// Mitsubishi GX Works2 project: BookEX3_1 POU   PLC: Q13UDV

TYPE CnvBlock : STRUCT
  bStartSW : BOOL;
  bEndSW : BOOL;
  BoxCnt : ARRAY [0..9] OF INT;
  sName : STRING[32];
  tOnDelay : TIME;
END_STRUCT END_TYPE

TYPE sdtLog : STRUCT
  idMonth : INT;
  idDay : INT;
  idHour : INT;
  idMin : INT;
  idSec : INT;
  idPID : DINT;
  wdData : ARRAY [0..39] OF INT;
  idYear : INT;
  idMsgNo : INT;
  idMsgLeng : INT;
END_STRUCT END_TYPE

TYPE ServoBlk : STRUCT
  RunCode : INT;
  ErrCode : INT;
  WarnCode : INT;
  ServoSts : WORD;
  CmdPos : DINT;
  CurrPos : DINT;
  CurrSp : INT;
  Torque : INT;
END_STRUCT END_TYPE

// global labels: Global
VAR_GLOBAL
  bVar0 AT M5000 : BOOL;
  abArray0 AT M5010 : ARRAY [0..49] OF BOOL;
  sStr0 AT D5000 : STRING[199];
  sStr1 AT D5100 : STRING[199];
  sStr2 AT D5200 : STRING[199];
  sStr3 AT D5300 : STRING[199];
  sStr4 AT D5400 : STRING[199];
  sStr5 AT D5500 : STRING[199];
  sStr6 AT D5600 : STRING[199];
  sStr7 AT D5700 : STRING[199];
  sStr8 AT D5800 : STRING[199];
  sStr9 AT D5900 : STRING[199];
  iVar0 AT D4500 : INT;
  iVar1 AT D4501 : INT;
  iVar2 AT D4502 : INT;
  iVar3 AT D4503 : INT;
  iVar4 AT D4504 : INT;
  iVar5 AT D4505 : INT;
  iVar6 AT D4506 : INT;
  iVar7 AT D4507 : INT;
  iVar8 AT D4508 : INT;
  iVar9 AT D4509 : INT;
  dVar0 AT D4510 : DINT;
  dVar1 AT D4512 : DINT;
  dVar2 AT D4514 : DINT;
  dVar3 AT D4516 : DINT;
  dVar4 AT D4518 : DINT;
  dVar5 AT D4520 : DINT;
  dVar6 AT D4522 : DINT;
  dVar7 AT D4524 : DINT;
  dVar8 AT D4526 : DINT;
  dVar9 AT D4528 : DINT;
  wVar0 AT D4530 : WORD;
  wVar1 AT D4531 : WORD;
  wVar2 AT D4532 : WORD;
  wVar3 AT D4533 : WORD;
  wVar4 AT D4534 : WORD;
  wVar5 AT D4535 : WORD;
  wVar6 AT D4536 : WORD;
  wVar7 AT D4537 : WORD;
  wVar8 AT D4538 : WORD;
  wVar9 AT D4539 : WORD;
  dwVar0 AT D4540 : DWORD;
  dwVar1 AT D4542 : DWORD;
  dwVar2 AT D4544 : DWORD;
  dwVar3 AT D4546 : DWORD;
  dwVar4 AT D4548 : DWORD;
  dwVar5 AT D4550 : DWORD;
  dwVar6 AT D4552 : DWORD;
  dwVar7 AT D4554 : DWORD;
  dwVar8 AT D4556 : DWORD;
  dwVar9 AT D4558 : DWORD;
  fsVar0 AT D4560 : REAL;
  fsVar1 AT D4562 : REAL;
  fsVar2 AT D4564 : REAL;
  fsVar3 AT D4566 : REAL;
  fsVar4 AT D4568 : REAL;
  fsVar5 AT D4570 : REAL;
  fsVar6 AT D4572 : REAL;
  fsVar7 AT D4574 : REAL;
  fsVar8 AT D4576 : REAL;
  fsVar9 AT D4578 : REAL;
  fdVar0 AT D4580 : LREAL;
  tTime0 AT D4620 : TIME;
  tTime1 AT D4622 : TIME;
  tTime2 AT D4624 : TIME;
  tTime3 AT D4626 : TIME;
  tTime4 AT D4628 : TIME;
  tTime5 AT D4630 : TIME;
  tTime6 AT D4632 : TIME;
  tTime7 AT D4634 : TIME;
  tTime8 AT D4636 : TIME;
  tTime9 AT D4638 : TIME;
  tTime10 AT D4640 : TIME;
  bVar1 AT M5001 : BOOL;
  bVar2 AT M5002 : BOOL;
  bVar3 AT M5003 : BOOL;
  bVar4 AT M5004 : BOOL;
  bVar5 AT M5005 : BOOL;
  bVar6 AT M5006 : BOOL;
  bVar7 AT M5007 : BOOL;
  bVar8 AT M5008 : BOOL;
  bVar9 AT M5009 : BOOL;
  abArray1 AT M5060 : ARRAY [0..49] OF BOOL;
  abArray2 AT M5110 : ARRAY [0..49] OF BOOL;
  abArray3 AT M5160 : ARRAY [0..49] OF BOOL;
  abArray4 AT M5210 : ARRAY [0..49] OF BOOL;
  abArray5 AT M5260 : ARRAY [0..49] OF BOOL;
  abArray6 AT M5310 : ARRAY [0..49] OF BOOL;
  abArray7 AT M5360 : ARRAY [0..49] OF BOOL;
  abArray8 AT M5410 : ARRAY [0..49] OF BOOL;
  abArray9 AT M5460 : ARRAY [0..49] OF BOOL;
  fdVar1 AT D4584 : LREAL;
  fdVar2 AT D4588 : LREAL;
  fdVar3 AT D4592 : LREAL;
  fdVar4 AT D4596 : LREAL;
  fdVar5 AT D4600 : LREAL;
  fdVar6 AT D4604 : LREAL;
  fdVar7 AT D4608 : LREAL;
  fdVar8 AT D4612 : LREAL;
  fdVar9 AT D4616 : LREAL;
  aSendData1 AT D100 : ARRAY [0..9] OF INT;
  aiTxData AT D4000 : ARRAY [0..99] OF INT;
  aiRxData AT D4100 : ARRAY [0..99] OF INT;
  iOpenOK AT D3900 : INT;
  iOpenERR AT D3901 : INT;
  iSendOK AT D3902 : INT;
  iSendERR AT D3903 : INT;
  iCloseOK AT D3906 : INT;
  iCloseERR AT D3907 : INT;
  iRecvOK AT D3904 : INT;
  iRecvERR AT D3905 : INT;
  aiTxData2 AT D4200 : ARRAY [0..99] OF INT;
  aiRxData2 AT D4300 : ARRAY [0..99] OF INT;
  iOpenOK2 AT D3908 : INT;
  iOpenERR2 AT D3909 : INT;
  iSendOK2 AT D3910 : INT;
  iSendERR2 AT D3911 : INT;
  iRecvOK2 AT D3912 : INT;
  iRecvERR2 AT D3913 : INT;
  iCloseOK2 AT D3914 : INT;
  iCloseERR2 AT D3915 : INT;
  iEOpenComp AT D3916 : INT;
  iEOpenReq AT D3917 : INT;
  iERecvFlag AT D3918 : INT;
  iOpenCode AT D3919 : INT;
  iSendCode AT D3920 : INT;
  iRecvCode AT D3921 : INT;
  iCloseCode AT D3922 : INT;
  iOpenCode2 AT D3923 : INT;
  iSendCode2 AT D3924 : INT;
  iRecvCode2 AT D3925 : INT;
  iCloseCode2 AT D3926 : INT;
  aRecvData1 AT D110 : ARRAY [0..9] OF INT;
  aSendData2 AT D120 : ARRAY [0..9] OF INT;
  aRecvData2 AT D130 : ARRAY [0..9] OF INT;
END_VAR
// user libraries (not included): HMI

PROGRAM ExPOU
VAR
  iNumber1 : ARRAY [0..9] OF INT;
  iNumber2 : ARRAY [0..9] OF INT;
  iNumber3 : ARRAY [0..9] OF INT;
  fbPytha_1 : fbPytha;
  fbPytha_2 : fbPytha;
  Function_Enable : BOOL;
  Enable_Out : BOOL;
END_VAR
(* structured ladder/FBD written out as ST: instructions are called as NAME(EN, inputs, outputs); _pN, _eN, _tN stand for wires *)
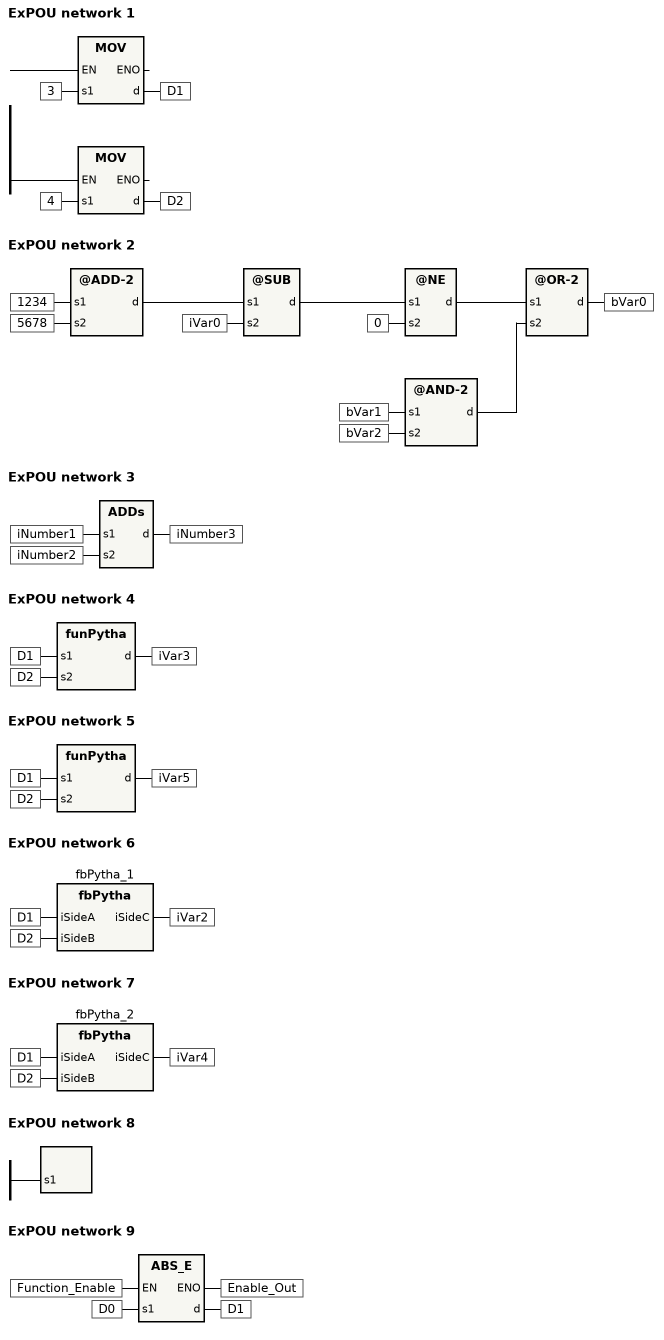
(* network 1 *)
MOV(TRUE, 3, D1);
MOV(TRUE, 4, D2);
(* network 2 *)
bVar0 := @OR-2(@NE(@SUB(@ADD-2(1234, 5678), iVar0), 0), @AND-2(bVar1, bVar2));
(* network 3 *)
iNumber3 := ADDs(iNumber1, iNumber2);
(* network 4 *)
iVar3 := funPytha(D1, D2);
(* network 5 *)
iVar5 := funPytha(D1, D2);
(* network 6 *)
fbPytha_1(iSideA := D1, iSideB := D2, iSideC => iVar2);
(* network 7 *)
fbPytha_2(iSideA := D1, iSideB := D2, iSideC => iVar4);
(* network 8 *)
(* element kind 10  <- TRUE *)
(* network 9 *)
_e1 := ABS_E(Function_Enable, D0, D1);
Enable_Out := _e1;
END_PROGRAM

FUNCTION ADDs
VAR_INPUT
  iInp1 : ARRAY [0..9] OF INT;
END_VAR
VAR
  ix : INT;
END_VAR
VAR_INPUT
  iInp2 : ARRAY [0..9] OF INT;
END_VAR
;
FOR ix := 0 TO 9 DO
	ADDs[ix] := iInp1[ix]+iInp2[ix];
END_FOR;
END_FUNCTION

FUNCTION_BLOCK fbPytha
VAR_INPUT
  iSideA : INT;
  iSideB : INT;
END_VAR
VAR_OUTPUT
  iSideC : INT;
END_VAR
VAR
  ix : INT;
  bBit1 : BOOL;
  bBit2 : BOOL;
  bBit3 : BOOL;
  bBit4 : BOOL;
  iInt1 : INT;
  iInt2 : INT;
  iInt3 : INT;
  iInt4 : INT;
  wWord1 : WORD;
  wWord2 : WORD;
  wWord3 : WORD;
  wWord4 : WORD;
END_VAR
;
iSideC := iSideA * iSideA + iSideB * iSideB;
(*
bBit1 := 2#01;
bBit2 := 8#01;
bBit3 := K1;
bBit4 := H1;

iInt1 := 2#111_000;
iInt2 := 8#111_000;
iInt3 := K1100;
iInt4 := 11_00;

wWord1 := 2#111_000;
wWord2 := 8#111_000;
wWord3 := 65535;
wWord4 := H1100;

fsVar0 := -2.34;
fsVar1 := E2.34;
fsVar2 := -2.34E-5;
fsVar3 := -2.34e6;
fsVar4 := 1.0;

tTime0 := T#1h;
tTime1 := T#1d2h3m4s5ms;
tTime2 := TIME#1h;

sStr0 := '가나다';
sStr1 := "ABC";
sStr2 := "가나다";
sStr3 := 'ABC';
 *)
END_FUNCTION_BLOCK

FUNCTION funPytha
VAR_INPUT
  iSideA : INT;
  iSideB : INT;
END_VAR
VAR
  ix : INT;
END_VAR
;
funPytha := iSideA * iSideA + iSideB * iSideB;
END_FUNCTION
